TYPE ST_ModuleCtrl :
STRUCT
	RequestId : UDINT;
	PackMLIn : ST_PML_Base_In;
	
	AlarmAckRequest : ST_AlarmAckRequest;
END_STRUCT
END_TYPE

(* stored: Version 1.1.0.1, ProductVersion 3.1.4026.18
   DUT ST_ModuleCtrl: Id {18a0c1b7-22ee-4ab8-bbd4-dc3f63dd976b} *)
